TYPE ST_Ampel_Zustand :
STRUCT
	Stellung_Rot		: BOOL;
	Stellung_Orange		: BOOL;
	Stellung_Gruen		: BOOL;
	Stellung_Blau		: BOOL;
	Stellung_Buzz		: BOOL;

	Stoerung			: BOOL;
	Stoerung_Code		: WORD;

	Warnung				: BOOL;
	Warnung_Code		: WORD;

	Status				: SINT;

	Quittierung			: BOOL;
END_STRUCT
END_TYPE

(* stored: Version 1.1.0.1, ProductVersion 3.1.4024.9
   DUT ST_Ampel_Zustand: Id {91cc7763-2e60-4fb6-9c1f-4e8f8f94302b} *)
